(* IEC 61131-3 sources: RL_MAR/experiments/comparison/autoplc/results/gpt-4o-mini_20260511_164212/hf_2, 1 file *)

(* ---- hf_2_1.st ---- *)
FUNCTION_BLOCK FindMinMaxValues
    VAR_INPUT
        values : ARRAY[1..10] OF DINT;
    END_VAR

    VAR_OUTPUT
        minValue : DINT;
        minValueIndex : DINT;
        maxValue : DINT;
        maxValueIndex : DINT;
    END_VAR

    VAR
        i : INT;
    END_VAR

    // Initialization
    minValue := values[1];
    maxValue := values[1];
    minValueIndex := 1;
    maxValueIndex := 1;

    // Iteration through the array
    FOR i := 1 TO 10 DO
        // Check for minimum value
        IF values[i] < minValue THEN
            minValue := values[i];
            minValueIndex := i;
        END_IF;

        // Check for maximum value
        IF values[i] > maxValue THEN
            maxValue := values[i];
            maxValueIndex := i;
        END_IF;
    END_FOR;
END_FUNCTION_BLOCK
